// TIA Portal V18 export
// export: Created 2026-01-09T11:32:10.846583Z, ExportSetting WithDefaults, DisplayName Totally Integrated Automation Portal, DisplayVersion V18 Update 5, DisplayName TIA Portal Openness, DisplayVersion V18 Update 5, DisplayName TIA Portal Teamcenter Gateway, DisplayVersion V18, DisplayName TIA Portal Version Control Interface, DisplayVersion V18, DisplayName SINAMICS Startdrive Advanced, DisplayVersion V18 SP2 Update 1, DisplayName SINAMICS Startdrive G110M, G120, G120C, G120D, G120P, G115D, DisplayVersion V18 SP2 Update 1, DisplayName SINAMICS Startdrive G130, G150, S120, S150, SINAMICS MV, S210, G220, S200, DisplayVersion V18 SP2 Update 1, DisplayName STEP 7 Professional, DisplayVersion V18 Update 5, DisplayName STEP 7 Safety, DisplayVersion V18, DisplayName WinCC Professional, DisplayVersion V18 Update 5
TagTable "Motor_1"
  MotorControl_Dev{1} : Motor_Control  (PLC tag MotorControl.Dev[1], CPU S71500-2PN_TP700, 1 s)
    TagStructureMember "Manual"
      TagStructureMember "Start"
      TagStructureMember "CCWStart"
      TagStructureMember "SpeedChange"
    TagStructureMember "Auto"
      TagStructureMember "Start"
      TagStructureMember "CCWStart"
      TagStructureMember "SpeedChange"
    TagStructureMember "OutControl"
      TagStructureMember "o_Start"
      TagStructureMember "o_CCWStart"
      TagStructureMember "o_SpeedChanged"
      TagStructureMember "o_Ready"
      TagStructureMember "o_Alarm"
    TagStructureMember "Error"
      TagArrayMember "[0]"
      TagArrayMember "[1]"
      TagArrayMember "[2]"
      TagArrayMember "[3]"
      TagArrayMember "[4]"
      TagArrayMember "[5]"
      TagArrayMember "[6]"
      TagArrayMember "[7]"
      TagArrayMember "[8]"
      TagArrayMember "[9]"
      TagArrayMember "[10]"
      TagArrayMember "[11]"
      TagArrayMember "[12]"
      TagArrayMember "[13]"
      TagArrayMember "[14]"
      TagArrayMember "[15]"
  MotorControl_Dev{2} : Motor_Control  (PLC tag MotorControl.Dev[2], CPU S71500-2PN_TP700, 1 s)
    TagStructureMember "Manual"
      TagStructureMember "Start"
      TagStructureMember "CCWStart"
      TagStructureMember "SpeedChange"
    TagStructureMember "Auto"
      TagStructureMember "Start"
      TagStructureMember "CCWStart"
      TagStructureMember "SpeedChange"
    TagStructureMember "OutControl"
      TagStructureMember "o_Start"
      TagStructureMember "o_CCWStart"
      TagStructureMember "o_SpeedChanged"
      TagStructureMember "o_Ready"
      TagStructureMember "o_Alarm"
    TagStructureMember "Error"
      TagArrayMember "[0]"
      TagArrayMember "[1]"
      TagArrayMember "[2]"
      TagArrayMember "[3]"
      TagArrayMember "[4]"
      TagArrayMember "[5]"
      TagArrayMember "[6]"
      TagArrayMember "[7]"
      TagArrayMember "[8]"
      TagArrayMember "[9]"
      TagArrayMember "[10]"
      TagArrayMember "[11]"
      TagArrayMember "[12]"
      TagArrayMember "[13]"
      TagArrayMember "[14]"
      TagArrayMember "[15]"
  MotorControl_Dev{3} : Motor_Control  (PLC tag MotorControl.Dev[3], CPU S71500-2PN_TP700, 1 s)
    TagStructureMember "Manual"
      TagStructureMember "Start"
      TagStructureMember "CCWStart"
      TagStructureMember "SpeedChange"
    TagStructureMember "Auto"
      TagStructureMember "Start"
      TagStructureMember "CCWStart"
      TagStructureMember "SpeedChange"
    TagStructureMember "OutControl"
      TagStructureMember "o_Start"
      TagStructureMember "o_CCWStart"
      TagStructureMember "o_SpeedChanged"
      TagStructureMember "o_Ready"
      TagStructureMember "o_Alarm"
    TagStructureMember "Error"
      TagArrayMember "[0]"
      TagArrayMember "[1]"
      TagArrayMember "[2]"
      TagArrayMember "[3]"
      TagArrayMember "[4]"
      TagArrayMember "[5]"
      TagArrayMember "[6]"
      TagArrayMember "[7]"
      TagArrayMember "[8]"
      TagArrayMember "[9]"
      TagArrayMember "[10]"
      TagArrayMember "[11]"
      TagArrayMember "[12]"
      TagArrayMember "[13]"
      TagArrayMember "[14]"
      TagArrayMember "[15]"
  MotorControl_Dev{4} : Motor_Control  (PLC tag MotorControl.Dev[4], CPU S71500-2PN_TP700, 1 s)
    TagStructureMember "Manual"
      TagStructureMember "Start"
      TagStructureMember "CCWStart"
      TagStructureMember "SpeedChange"
    TagStructureMember "Auto"
      TagStructureMember "Start"
      TagStructureMember "CCWStart"
      TagStructureMember "SpeedChange"
    TagStructureMember "OutControl"
      TagStructureMember "o_Start"
      TagStructureMember "o_CCWStart"
      TagStructureMember "o_SpeedChanged"
      TagStructureMember "o_Ready"
      TagStructureMember "o_Alarm"
    TagStructureMember "Error"
      TagArrayMember "[0]"
      TagArrayMember "[1]"
      TagArrayMember "[2]"
      TagArrayMember "[3]"
      TagArrayMember "[4]"
      TagArrayMember "[5]"
      TagArrayMember "[6]"
      TagArrayMember "[7]"
      TagArrayMember "[8]"
      TagArrayMember "[9]"
      TagArrayMember "[10]"
      TagArrayMember "[11]"
      TagArrayMember "[12]"
      TagArrayMember "[13]"
      TagArrayMember "[14]"
      TagArrayMember "[15]"
  MotorControl_Dev{5} : Motor_Control  (PLC tag MotorControl.Dev[5], CPU S71500-2PN_TP700, 1 s)
    TagStructureMember "Manual"
      TagStructureMember "Start"
      TagStructureMember "CCWStart"
      TagStructureMember "SpeedChange"
    TagStructureMember "Auto"
      TagStructureMember "Start"
      TagStructureMember "CCWStart"
      TagStructureMember "SpeedChange"
    TagStructureMember "OutControl"
      TagStructureMember "o_Start"
      TagStructureMember "o_CCWStart"
      TagStructureMember "o_SpeedChanged"
      TagStructureMember "o_Ready"
      TagStructureMember "o_Alarm"
    TagStructureMember "Error"
      TagArrayMember "[0]"
      TagArrayMember "[1]"
      TagArrayMember "[2]"
      TagArrayMember "[3]"
      TagArrayMember "[4]"
      TagArrayMember "[5]"
      TagArrayMember "[6]"
      TagArrayMember "[7]"
      TagArrayMember "[8]"
      TagArrayMember "[9]"
      TagArrayMember "[10]"
      TagArrayMember "[11]"
      TagArrayMember "[12]"
      TagArrayMember "[13]"
      TagArrayMember "[14]"
      TagArrayMember "[15]"
  MotorControl_Dev{6} : Motor_Control  (PLC tag MotorControl.Dev[6], CPU S71500-2PN_TP700, 1 s)
    TagStructureMember "Manual"
      TagStructureMember "Start"
      TagStructureMember "CCWStart"
      TagStructureMember "SpeedChange"
    TagStructureMember "Auto"
      TagStructureMember "Start"
      TagStructureMember "CCWStart"
      TagStructureMember "SpeedChange"
    TagStructureMember "OutControl"
      TagStructureMember "o_Start"
      TagStructureMember "o_CCWStart"
      TagStructureMember "o_SpeedChanged"
      TagStructureMember "o_Ready"
      TagStructureMember "o_Alarm"
    TagStructureMember "Error"
      TagArrayMember "[0]"
      TagArrayMember "[1]"
      TagArrayMember "[2]"
      TagArrayMember "[3]"
      TagArrayMember "[4]"
      TagArrayMember "[5]"
      TagArrayMember "[6]"
      TagArrayMember "[7]"
      TagArrayMember "[8]"
      TagArrayMember "[9]"
      TagArrayMember "[10]"
      TagArrayMember "[11]"
      TagArrayMember "[12]"
      TagArrayMember "[13]"
      TagArrayMember "[14]"
      TagArrayMember "[15]"
  MotorControl_Dev{7} : Motor_Control  (PLC tag MotorControl.Dev[7], CPU S71500-2PN_TP700, 1 s)
    TagStructureMember "Manual"
      TagStructureMember "Start"
      TagStructureMember "CCWStart"
      TagStructureMember "SpeedChange"
    TagStructureMember "Auto"
      TagStructureMember "Start"
      TagStructureMember "CCWStart"
      TagStructureMember "SpeedChange"
    TagStructureMember "OutControl"
      TagStructureMember "o_Start"
      TagStructureMember "o_CCWStart"
      TagStructureMember "o_SpeedChanged"
      TagStructureMember "o_Ready"
      TagStructureMember "o_Alarm"
    TagStructureMember "Error"
      TagArrayMember "[0]"
      TagArrayMember "[1]"
      TagArrayMember "[2]"
      TagArrayMember "[3]"
      TagArrayMember "[4]"
      TagArrayMember "[5]"
      TagArrayMember "[6]"
      TagArrayMember "[7]"
      TagArrayMember "[8]"
      TagArrayMember "[9]"
      TagArrayMember "[10]"
      TagArrayMember "[11]"
      TagArrayMember "[12]"
      TagArrayMember "[13]"
      TagArrayMember "[14]"
      TagArrayMember "[15]"
  MotorControl_Dev{8} : Motor_Control  (PLC tag MotorControl.Dev[8], CPU S71500-2PN_TP700, 1 s)
    TagStructureMember "Manual"
      TagStructureMember "Start"
      TagStructureMember "CCWStart"
      TagStructureMember "SpeedChange"
    TagStructureMember "Auto"
      TagStructureMember "Start"
      TagStructureMember "CCWStart"
      TagStructureMember "SpeedChange"
    TagStructureMember "OutControl"
      TagStructureMember "o_Start"
      TagStructureMember "o_CCWStart"
      TagStructureMember "o_SpeedChanged"
      TagStructureMember "o_Ready"
      TagStructureMember "o_Alarm"
    TagStructureMember "Error"
      TagArrayMember "[0]"
      TagArrayMember "[1]"
      TagArrayMember "[2]"
      TagArrayMember "[3]"
      TagArrayMember "[4]"
      TagArrayMember "[5]"
      TagArrayMember "[6]"
      TagArrayMember "[7]"
      TagArrayMember "[8]"
      TagArrayMember "[9]"
      TagArrayMember "[10]"
      TagArrayMember "[11]"
      TagArrayMember "[12]"
      TagArrayMember "[13]"
      TagArrayMember "[14]"
      TagArrayMember "[15]"
  MotorControl_Dev{9} : Motor_Control  (PLC tag MotorControl.Dev[9], CPU S71500-2PN_TP700, 1 s)
    TagStructureMember "Manual"
      TagStructureMember "Start"
      TagStructureMember "CCWStart"
      TagStructureMember "SpeedChange"
    TagStructureMember "Auto"
      TagStructureMember "Start"
      TagStructureMember "CCWStart"
      TagStructureMember "SpeedChange"
    TagStructureMember "OutControl"
      TagStructureMember "o_Start"
      TagStructureMember "o_CCWStart"
      TagStructureMember "o_SpeedChanged"
      TagStructureMember "o_Ready"
      TagStructureMember "o_Alarm"
    TagStructureMember "Error"
      TagArrayMember "[0]"
      TagArrayMember "[1]"
      TagArrayMember "[2]"
      TagArrayMember "[3]"
      TagArrayMember "[4]"
      TagArrayMember "[5]"
      TagArrayMember "[6]"
      TagArrayMember "[7]"
      TagArrayMember "[8]"
      TagArrayMember "[9]"
      TagArrayMember "[10]"
      TagArrayMember "[11]"
      TagArrayMember "[12]"
      TagArrayMember "[13]"
      TagArrayMember "[14]"
      TagArrayMember "[15]"
  MotorControl_Dev{10} : Motor_Control  (PLC tag MotorControl.Dev[10], CPU S71500-2PN_TP700, 1 s)
    TagStructureMember "Manual"
      TagStructureMember "Start"
      TagStructureMember "CCWStart"
      TagStructureMember "SpeedChange"
    TagStructureMember "Auto"
      TagStructureMember "Start"
      TagStructureMember "CCWStart"
      TagStructureMember "SpeedChange"
    TagStructureMember "OutControl"
      TagStructureMember "o_Start"
      TagStructureMember "o_CCWStart"
      TagStructureMember "o_SpeedChanged"
      TagStructureMember "o_Ready"
      TagStructureMember "o_Alarm"
    TagStructureMember "Error"
      TagArrayMember "[0]"
      TagArrayMember "[1]"
      TagArrayMember "[2]"
      TagArrayMember "[3]"
      TagArrayMember "[4]"
      TagArrayMember "[5]"
      TagArrayMember "[6]"
      TagArrayMember "[7]"
      TagArrayMember "[8]"
      TagArrayMember "[9]"
      TagArrayMember "[10]"
      TagArrayMember "[11]"
      TagArrayMember "[12]"
      TagArrayMember "[13]"
      TagArrayMember "[14]"
      TagArrayMember "[15]"
  MotorControl_Dev{11} : Motor_Control  (PLC tag MotorControl.Dev[11], CPU S71500-2PN_TP700, 1 s)
    TagStructureMember "Manual"
      TagStructureMember "Start"
      TagStructureMember "CCWStart"
      TagStructureMember "SpeedChange"
    TagStructureMember "Auto"
      TagStructureMember "Start"
      TagStructureMember "CCWStart"
      TagStructureMember "SpeedChange"
    TagStructureMember "OutControl"
      TagStructureMember "o_Start"
      TagStructureMember "o_CCWStart"
      TagStructureMember "o_SpeedChanged"
      TagStructureMember "o_Ready"
      TagStructureMember "o_Alarm"
    TagStructureMember "Error"
      TagArrayMember "[0]"
      TagArrayMember "[1]"
      TagArrayMember "[2]"
      TagArrayMember "[3]"
      TagArrayMember "[4]"
      TagArrayMember "[5]"
      TagArrayMember "[6]"
      TagArrayMember "[7]"
      TagArrayMember "[8]"
      TagArrayMember "[9]"
      TagArrayMember "[10]"
      TagArrayMember "[11]"
      TagArrayMember "[12]"
      TagArrayMember "[13]"
      TagArrayMember "[14]"
      TagArrayMember "[15]"
  MotorControl_Dev{12} : Motor_Control  (PLC tag MotorControl.Dev[12], CPU S71500-2PN_TP700, 1 s)
    TagStructureMember "Manual"
      TagStructureMember "Start"
      TagStructureMember "CCWStart"
      TagStructureMember "SpeedChange"
    TagStructureMember "Auto"
      TagStructureMember "Start"
      TagStructureMember "CCWStart"
      TagStructureMember "SpeedChange"
    TagStructureMember "OutControl"
      TagStructureMember "o_Start"
      TagStructureMember "o_CCWStart"
      TagStructureMember "o_SpeedChanged"
      TagStructureMember "o_Ready"
      TagStructureMember "o_Alarm"
    TagStructureMember "Error"
      TagArrayMember "[0]"
      TagArrayMember "[1]"
      TagArrayMember "[2]"
      TagArrayMember "[3]"
      TagArrayMember "[4]"
      TagArrayMember "[5]"
      TagArrayMember "[6]"
      TagArrayMember "[7]"
      TagArrayMember "[8]"
      TagArrayMember "[9]"
      TagArrayMember "[10]"
      TagArrayMember "[11]"
      TagArrayMember "[12]"
      TagArrayMember "[13]"
      TagArrayMember "[14]"
      TagArrayMember "[15]"
  MotorControl_Dev{13} : Motor_Control  (PLC tag MotorControl.Dev[13], CPU S71500-2PN_TP700, 1 s)
    TagStructureMember "Manual"
      TagStructureMember "Start"
      TagStructureMember "CCWStart"
      TagStructureMember "SpeedChange"
    TagStructureMember "Auto"
      TagStructureMember "Start"
      TagStructureMember "CCWStart"
      TagStructureMember "SpeedChange"
    TagStructureMember "OutControl"
      TagStructureMember "o_Start"
      TagStructureMember "o_CCWStart"
      TagStructureMember "o_SpeedChanged"
      TagStructureMember "o_Ready"
      TagStructureMember "o_Alarm"
    TagStructureMember "Error"
      TagArrayMember "[0]"
      TagArrayMember "[1]"
      TagArrayMember "[2]"
      TagArrayMember "[3]"
      TagArrayMember "[4]"
      TagArrayMember "[5]"
      TagArrayMember "[6]"
      TagArrayMember "[7]"
      TagArrayMember "[8]"
      TagArrayMember "[9]"
      TagArrayMember "[10]"
      TagArrayMember "[11]"
      TagArrayMember "[12]"
      TagArrayMember "[13]"
      TagArrayMember "[14]"
      TagArrayMember "[15]"
  MotorControl_Dev{14} : Motor_Control  (PLC tag MotorControl.Dev[14], CPU S71500-2PN_TP700, 1 s)
    TagStructureMember "Manual"
      TagStructureMember "Start"
      TagStructureMember "CCWStart"
      TagStructureMember "SpeedChange"
    TagStructureMember "Auto"
      TagStructureMember "Start"
      TagStructureMember "CCWStart"
      TagStructureMember "SpeedChange"
    TagStructureMember "OutControl"
      TagStructureMember "o_Start"
      TagStructureMember "o_CCWStart"
      TagStructureMember "o_SpeedChanged"
      TagStructureMember "o_Ready"
      TagStructureMember "o_Alarm"
    TagStructureMember "Error"
      TagArrayMember "[0]"
      TagArrayMember "[1]"
      TagArrayMember "[2]"
      TagArrayMember "[3]"
      TagArrayMember "[4]"
      TagArrayMember "[5]"
      TagArrayMember "[6]"
      TagArrayMember "[7]"
      TagArrayMember "[8]"
      TagArrayMember "[9]"
      TagArrayMember "[10]"
      TagArrayMember "[11]"
      TagArrayMember "[12]"
      TagArrayMember "[13]"
      TagArrayMember "[14]"
      TagArrayMember "[15]"
  MotorControl_Dev{15} : Motor_Control  (PLC tag MotorControl.Dev[15], CPU S71500-2PN_TP700, 1 s)
    TagStructureMember "Manual"
      TagStructureMember "Start"
      TagStructureMember "CCWStart"
      TagStructureMember "SpeedChange"
    TagStructureMember "Auto"
      TagStructureMember "Start"
      TagStructureMember "CCWStart"
      TagStructureMember "SpeedChange"
    TagStructureMember "OutControl"
      TagStructureMember "o_Start"
      TagStructureMember "o_CCWStart"
      TagStructureMember "o_SpeedChanged"
      TagStructureMember "o_Ready"
      TagStructureMember "o_Alarm"
    TagStructureMember "Error"
      TagArrayMember "[0]"
      TagArrayMember "[1]"
      TagArrayMember "[2]"
      TagArrayMember "[3]"
      TagArrayMember "[4]"
      TagArrayMember "[5]"
      TagArrayMember "[6]"
      TagArrayMember "[7]"
      TagArrayMember "[8]"
      TagArrayMember "[9]"
      TagArrayMember "[10]"
      TagArrayMember "[11]"
      TagArrayMember "[12]"
      TagArrayMember "[13]"
      TagArrayMember "[14]"
      TagArrayMember "[15]"
  MotorControl_Dev{16} : Motor_Control  (PLC tag MotorControl.Dev[16], CPU S71500-2PN_TP700, 1 s)
    TagStructureMember "Manual"
      TagStructureMember "Start"
      TagStructureMember "CCWStart"
      TagStructureMember "SpeedChange"
    TagStructureMember "Auto"
      TagStructureMember "Start"
      TagStructureMember "CCWStart"
      TagStructureMember "SpeedChange"
    TagStructureMember "OutControl"
      TagStructureMember "o_Start"
      TagStructureMember "o_CCWStart"
      TagStructureMember "o_SpeedChanged"
      TagStructureMember "o_Ready"
      TagStructureMember "o_Alarm"
    TagStructureMember "Error"
      TagArrayMember "[0]"
      TagArrayMember "[1]"
      TagArrayMember "[2]"
      TagArrayMember "[3]"
      TagArrayMember "[4]"
      TagArrayMember "[5]"
      TagArrayMember "[6]"
      TagArrayMember "[7]"
      TagArrayMember "[8]"
      TagArrayMember "[9]"
      TagArrayMember "[10]"
      TagArrayMember "[11]"
      TagArrayMember "[12]"
      TagArrayMember "[13]"
      TagArrayMember "[14]"
      TagArrayMember "[15]"
  MotorControl_Dev{17} : Motor_Control  (PLC tag MotorControl.Dev[17], CPU S71500-2PN_TP700, 1 s)
    TagStructureMember "Manual"
      TagStructureMember "Start"
      TagStructureMember "CCWStart"
      TagStructureMember "SpeedChange"
    TagStructureMember "Auto"
      TagStructureMember "Start"
      TagStructureMember "CCWStart"
      TagStructureMember "SpeedChange"
    TagStructureMember "OutControl"
      TagStructureMember "o_Start"
      TagStructureMember "o_CCWStart"
      TagStructureMember "o_SpeedChanged"
      TagStructureMember "o_Ready"
      TagStructureMember "o_Alarm"
    TagStructureMember "Error"
      TagArrayMember "[0]"
      TagArrayMember "[1]"
      TagArrayMember "[2]"
      TagArrayMember "[3]"
      TagArrayMember "[4]"
      TagArrayMember "[5]"
      TagArrayMember "[6]"
      TagArrayMember "[7]"
      TagArrayMember "[8]"
      TagArrayMember "[9]"
      TagArrayMember "[10]"
      TagArrayMember "[11]"
      TagArrayMember "[12]"
      TagArrayMember "[13]"
      TagArrayMember "[14]"
      TagArrayMember "[15]"
  MotorControl_Dev{18} : Motor_Control  (PLC tag MotorControl.Dev[18], CPU S71500-2PN_TP700, 1 s)
    TagStructureMember "Manual"
      TagStructureMember "Start"
      TagStructureMember "CCWStart"
      TagStructureMember "SpeedChange"
    TagStructureMember "Auto"
      TagStructureMember "Start"
      TagStructureMember "CCWStart"
      TagStructureMember "SpeedChange"
    TagStructureMember "OutControl"
      TagStructureMember "o_Start"
      TagStructureMember "o_CCWStart"
      TagStructureMember "o_SpeedChanged"
      TagStructureMember "o_Ready"
      TagStructureMember "o_Alarm"
    TagStructureMember "Error"
      TagArrayMember "[0]"
      TagArrayMember "[1]"
      TagArrayMember "[2]"
      TagArrayMember "[3]"
      TagArrayMember "[4]"
      TagArrayMember "[5]"
      TagArrayMember "[6]"
      TagArrayMember "[7]"
      TagArrayMember "[8]"
      TagArrayMember "[9]"
      TagArrayMember "[10]"
      TagArrayMember "[11]"
      TagArrayMember "[12]"
      TagArrayMember "[13]"
      TagArrayMember "[14]"
      TagArrayMember "[15]"
  MotorControl_Dev{19} : Motor_Control  (PLC tag MotorControl.Dev[19], CPU S71500-2PN_TP700, 1 s)
    TagStructureMember "Manual"
      TagStructureMember "Start"
      TagStructureMember "CCWStart"
      TagStructureMember "SpeedChange"
    TagStructureMember "Auto"
      TagStructureMember "Start"
      TagStructureMember "CCWStart"
      TagStructureMember "SpeedChange"
    TagStructureMember "OutControl"
      TagStructureMember "o_Start"
      TagStructureMember "o_CCWStart"
      TagStructureMember "o_SpeedChanged"
      TagStructureMember "o_Ready"
      TagStructureMember "o_Alarm"
    TagStructureMember "Error"
      TagArrayMember "[0]"
      TagArrayMember "[1]"
      TagArrayMember "[2]"
      TagArrayMember "[3]"
      TagArrayMember "[4]"
      TagArrayMember "[5]"
      TagArrayMember "[6]"
      TagArrayMember "[7]"
      TagArrayMember "[8]"
      TagArrayMember "[9]"
      TagArrayMember "[10]"
      TagArrayMember "[11]"
      TagArrayMember "[12]"
      TagArrayMember "[13]"
      TagArrayMember "[14]"
      TagArrayMember "[15]"
  MotorControl_Dev{20} : Motor_Control  (PLC tag MotorControl.Dev[20], CPU S71500-2PN_TP700, 1 s)
    TagStructureMember "Manual"
      TagStructureMember "Start"
      TagStructureMember "CCWStart"
      TagStructureMember "SpeedChange"
    TagStructureMember "Auto"
      TagStructureMember "Start"
      TagStructureMember "CCWStart"
      TagStructureMember "SpeedChange"
    TagStructureMember "OutControl"
      TagStructureMember "o_Start"
      TagStructureMember "o_CCWStart"
      TagStructureMember "o_SpeedChanged"
      TagStructureMember "o_Ready"
      TagStructureMember "o_Alarm"
    TagStructureMember "Error"
      TagArrayMember "[0]"
      TagArrayMember "[1]"
      TagArrayMember "[2]"
      TagArrayMember "[3]"
      TagArrayMember "[4]"
      TagArrayMember "[5]"
      TagArrayMember "[6]"
      TagArrayMember "[7]"
      TagArrayMember "[8]"
      TagArrayMember "[9]"
      TagArrayMember "[10]"
      TagArrayMember "[11]"
      TagArrayMember "[12]"
      TagArrayMember "[13]"
      TagArrayMember "[14]"
      TagArrayMember "[15]"
